{attribute 'GeneratedUsingTerminal: EL5101--0000'}
{attribute addProperty BoxType "EL5101--0000"}
{attribute addProperty Id "CtrlAT %Q*USINT1ValueAT %Q*UINT2"}
{attribute addProperty CRC "3329760021"}
{attribute addProperty Size "3"}
TYPE Channel_C6781B15 :
STRUCT
	{attribute addProperty Name "Ctrl"}
	Ctrl AT %Q* : USINT;
	{attribute addProperty Name "Value"}
	Value AT %Q* : UINT;
END_STRUCT
END_TYPE

(* stored: Version 1.2.0.0, ProductVersion 3.1.4024.9
   DUT Channel_C6781B15: Id {72931e0e-3299-4af5-aa04-31f754a88046} *)
